PROGRAM Timers
VAR
	SecondsTimer: Timer;
	LastTime, Now: LINT;
	InitDone: BOOL;
	BlinkPeriod: INT;
	CurrentBlinkPeriod: INT;
END_VAR

IF NOT InitDone THEN
	Now := SecondsTimer.ElapsedTime();
	InitDone := TRUE;
END_IF

// Show that we are alive
Globals.LifeCounter := Globals.LifeCounter + 1;

// Count seconds
Globals.SecondsCounter := SecondsTimer.ElapsedTime() / 1000;

IF Main.GreenMaster.VentilationRunning THEN
	IF Main.GreenMaster.TemperatureControlRunning THEN
		BlinkPeriod := 250;
	ELSE
		BlinkPeriod := 1000;
	END_IF
ELSE
	BlinkPeriod := 3000;
END_IF

IF BlinkPeriod <> CurrentBlinkPeriod THEN
	LastTime := SecondsTimer.ElapsedTime();
END_IF

IF Main.GreenMaster.Parameters.System.Operation.EN THEN
	// Blink ERR LED
	Now := SecondsTimer.ElapsedTime();
	IF (Now - LastTime) > (BlinkPeriod - 50) THEN
		F_CX8190_LED_ERR(eMode := E_CX81x0_LED.eCX81x0_LED_GREEN_ON);
	END_IF
	IF (Now - LastTime) > BlinkPeriod THEN
		F_CX8190_LED_ERR(eMode := E_CX81x0_LED.eCX81x0_LED_GREEN_OFF);
		LastTime := LastTime + BlinkPeriod; 
	END_IF
ELSE
	F_CX8190_LED_ERR(eMode := E_CX81x0_LED.eCX81x0_LED_RED_ON);
END_IF
CurrentBlinkPeriod := BlinkPeriod;

END_PROGRAM

(* stored: Version 1.1.0.1, ProductVersion 3.1.4024.6
   POU Timers: Id {6c48a0e3-a487-49da-89e6-6324bbaf0e4b}, SpecialFunc None *)
